FUNCTION_BLOCK FB_CONCAT (* Concatenation of WSTRING inputs *)
  (* Standard: 61499-1 *)
  (* Version 0.1, 2004-06-23, JHC, Rockwell Automation, Moved from fb.rt.diag to fb.rt.math. *)
  (* Version 0.0, 2001-04-12, JHC, Rockwell Automation, First XML version. *)
  (* Compiler header: package fb.rt.math; *)
  (* Compiler Java Sun JDK 1.4.2 *)
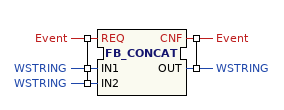
  EVENT_INPUT
    REQ WITH IN1, IN2;
  END_EVENT
  EVENT_OUTPUT
    CNF WITH OUT;
  END_EVENT
  VAR_INPUT
    IN1 : WSTRING;
    IN2 : WSTRING;
  END_VAR
  VAR_OUTPUT
    OUT : WSTRING;
  END_VAR
  ALGORITHM REQ IN Java:
OUT.value=IN1.value+IN2.value;
CNF.serviceEvent(this);
  END_ALGORITHM
END_FUNCTION_BLOCK
